//{attribute 'qualified_only'}
VAR_GLOBAL
END_VAR
VAR_GLOBAL CONSTANT
	gSystemTimeMaxNum		:UINT:=2000;// systemTimeModule 计时器数组最大值 最大值为2000
END_VAR

(* stored: Version 1.1.0.1, ProductVersion 3.1.4024.4
   GVL GVL_SystemTimeModule: Id {0f02fb37-c895-4af3-9868-b8420a6dd8a1} *)
